// TIA Portal V20 export
TYPE "MOVIMOT_Datos"
   STRUCT
      ENABLE : Bool;
      RESET : Bool;
      BRAKE_RELEASE : Bool;   // without_ENABLE
      "SPEED%" : Int;
      RAMP : Int := 1000;
      READY : Bool;
      FAULT : Bool;
      ERROR_NO : Int;
      CURRENT : Int;
   END_STRUCT;
END_TYPE
